// TIA Portal project "Trafik Işıkları Uygulaması 1" (V17)

(* hardware
DEVICE "S71500/ET200MP-Station_1"  S7-1500 station
   slot 0: "Profilschiene_0"  Rack  6ES7 590-1***0-0AA0
   slot 1: "PLC_1"  CPU 1518-4 PN/DP  6ES7 518-4AP00-0AB0  V2.9
      slot 3: "CPU-Display_1"  6ES7591-1BA00-0AA0
      slot 32768: "PROFINET-Schnittstelle_1"  X1
         slot 32769: "Port_1"  X1 P1
         slot 32770: "Port_2"  X1 P2
      slot 33024: "PROFINET interface_1"  X2
      slot 33280: "PROFINET interface GBIT_3"  X3
      slot 33536: "DP interface_1"  X4
      slot 34817: "Virtual CP interface port_1"  Virtual CP interface port  Virtual CP interface port
   slot 2: "AI 8xU/I/RTD/TC ST_1"  AI 8xU/I/RTD/TC ST  6ES7 531-7KF00-0AB0  V2.0
   slot 3: "AI 8xU/I/RTD/TC ST_2"  AI 8xU/I/RTD/TC ST  6ES7 531-7KF00-0AB0  V2.0
   slot 4: "AI 8xU/I/RTD/TC ST_3"  AI 8xU/I/RTD/TC ST  6ES7 531-7KF00-0AB0  V2.0
   slot 5: "AI 8xU/I/RTD/TC ST_4"  AI 8xU/I/RTD/TC ST  6ES7 531-7KF00-0AB0  V2.0
   slot 6: "DI 16x24VDC BA_1"  DI 16x24VDC BA  6ES7 521-1BH10-0AA0  V1.0
*)

// ===== PLC "PLC_1"  CPU 1518-4 PN/DP =====

VAR_GLOBAL   // PLC tag table "Standard-Variablentabelle"
   "START" AT %E0.0 : Bool;
   "A KIRMIZI" AT %A0.0 : Bool;
   "BAKIM" AT %E0.1 : Bool;
   "YARDIMCI KONTAK" AT %M0.0 : Bool;
   "Tag_2" AT %I0.2 : Bool;
   "DÖNGÜ" AT %M0.1 : Bool;
   "Tag_4" AT %T1 : Timer;
   "A SARI" AT %Q0.1 : Bool;
   "A YESİL" AT %Q0.2 : Bool;
   "B YESİL" AT %Q0.5 : Bool;
   "A YAYA Y" AT %Q0.7 : Bool;
   "B YAYA K" AT %Q1.0 : Bool;
   "B SARI" AT %Q0.4 : Bool;
   "B KIRMIZI" AT %Q0.3 : Bool;
   "B YAYA Y" AT %Q1.1 : Bool;
   "A YAYA K" AT %Q0.6 : Bool;
   "BAKIM YARDIMCI KONTAK" AT %M0.2 : Bool;
   "Clock_Byte" AT %MB50 : Byte;
   "Clock_10Hz" AT %M50.0 : Bool;
   "Clock_5Hz" AT %M50.1 : Bool;
   "Clock_2.5Hz" AT %M50.2 : Bool;
   "Clock_2Hz" AT %M50.3 : Bool;
   "Clock_1.25Hz" AT %M50.4 : Bool;
   "Clock_1Hz" AT %M50.5 : Bool;
   "Clock_0.625Hz" AT %M50.6 : Bool;
   "Clock_0.5Hz" AT %M50.7 : Bool;
   "Tag_1" AT %MD30 : Time;
   "Işık Süre" AT %QD30 : Time;
   "Tag_3" AT %QW30 : Word;
   "Tag_5" AT %MW30 : Word;
   "Tag_6" AT %ID30 : Time;
END_VAR

// folder: System blocks/Program resources

DATA_BLOCK "T1"   // DB1
{ S7_Optimized_Access := 'TRUE' }
AUTHOR : Simatic
FAMILY : IEC
NAME : IEC_TMR
VERSION : 1.0
// stored: InstanceOfName IEC_TIMER
"IEC_TIMER"
BEGIN
END_DATA_BLOCK

DATA_BLOCK "T2"   // DB2
{ S7_Optimized_Access := 'TRUE' }
AUTHOR : Simatic
FAMILY : IEC
NAME : IEC_TMR
VERSION : 1.0
// stored: InstanceOfName IEC_TIMER
"IEC_TIMER"
BEGIN
END_DATA_BLOCK

DATA_BLOCK "T3"   // DB3
{ S7_Optimized_Access := 'TRUE' }
AUTHOR : Simatic
FAMILY : IEC
NAME : IEC_TMR
VERSION : 1.0
// stored: InstanceOfName IEC_TIMER
"IEC_TIMER"
BEGIN
END_DATA_BLOCK

DATA_BLOCK "T4"   // DB5
{ S7_Optimized_Access := 'TRUE' }
AUTHOR : Simatic
FAMILY : IEC
NAME : IEC_TMR
VERSION : 1.0
// stored: InstanceOfName IEC_TIMER
"IEC_TIMER"
BEGIN
END_DATA_BLOCK

// folder: (top level)

FUNCTION "MHJ-PLC-Lab-Function-S71500" : Void   // FC9000, SCL
{ S7_Optimized_Access := 'TRUE' }
VERSION : 0.1
   VAR_TEMP
      Value : Byte;
      ForCounter : Int;
   END_VAR
   VAR CONSTANT
      Value_01_DW : DWord := 16#1223_5486;
      Value_02_DW : DWord := 16#A6C9_D1F5;
   END_VAR
BEGIN

   #Value:=PEEK(area := 16#82,
        dbNumber := 0,
        byteOffset := 511);
   #Value := #Value + 1;

   POKE(area := 16#82,
        dbNumber := 0,
        byteOffset := 511,
        value := #Value);

   POKE(area := 16#82,
        dbNumber := 0,
        byteOffset := 1016,
        value := #Value_01_DW);
   POKE(area := 16#82,
        dbNumber := 0,
        byteOffset := 1020,
        value := #Value_02_DW);

   FOR #ForCounter := 0 TO 63 DO
       #Value:=PEEK(area := 16#1,
            dbNumber := 0,
            byteOffset := #ForCounter);
       POKE(area := 16#81,
            dbNumber := 0,
            byteOffset := #ForCounter,
            value := #Value);
   END_FOR;
   #Value := PEEK(area := 16#1,
                  dbNumber := 0,
                  byteOffset := 512);
   POKE(area := 16#82,
        dbNumber := 0,
        byteOffset := 512,
        value := #Value);
END_FUNCTION

ORGANIZATION_BLOCK "Main"   // OB1, LAD, ProgramCycle
TITLE = "Main Program Sweep (Cycle)"
{ S7_Optimized_Access := 'TRUE' }
VERSION : 0.1
   VAR_INPUT
      Initial_Call : Bool;   // Initial call of this OB
      Remanence : Bool;   // =True, if remanent data are available
   END_VAR
   VAR_TEMP   // added for the SCL form of the ladder/FBD networks
      _w1 : Bool;
   END_VAR
BEGIN

REGION Network 1
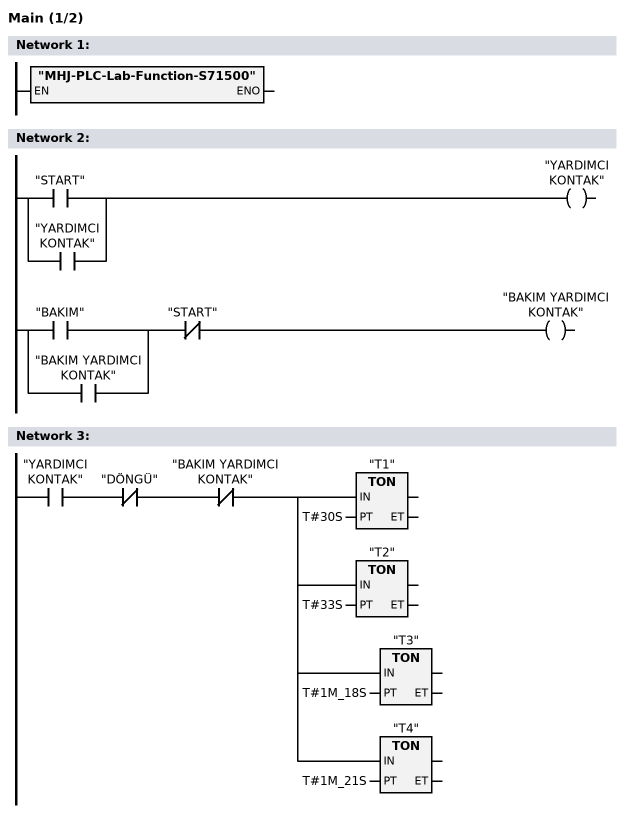
   RUNG wire#powerrail
      "MHJ-PLC-Lab-Function-S71500"()
   END_RUNG
   // the same network as SCL:
   "MHJ-PLC-Lab-Function-S71500"();
END_REGION

REGION Network 2
   RUNG wire#powerrail
      Contact( "START" )
      wire#w1
      Coil( "YARDIMCI KONTAK" )
   END_RUNG
   RUNG wire#powerrail
      Contact( "YARDIMCI KONTAK" )
   END_RUNG wire#w1
   RUNG wire#powerrail
      Contact( "BAKIM" )
      wire#w2
      I_Contact( "START" )
      Coil( "BAKIM YARDIMCI KONTAK" )
   END_RUNG
   RUNG wire#powerrail
      Contact( "BAKIM YARDIMCI KONTAK" )
   END_RUNG wire#w2
   // the same network as SCL:
   "YARDIMCI KONTAK" := "START" OR "YARDIMCI KONTAK";
   "BAKIM YARDIMCI KONTAK" := ("BAKIM" OR "BAKIM YARDIMCI KONTAK") AND NOT "START";
END_REGION

REGION Network 3
   #_w1 := "YARDIMCI KONTAK" AND NOT "DÖNGÜ" AND NOT "BAKIM YARDIMCI KONTAK";
   "T1".TON(IN := #_w1, PT := T#30S);
   "T2".TON(IN := #_w1, PT := T#33S);
   "T3".TON(IN := #_w1, PT := T#1M_18S);
   "T4".TON(IN := #_w1, PT := T#1M_21S);
END_REGION

REGION Network 4
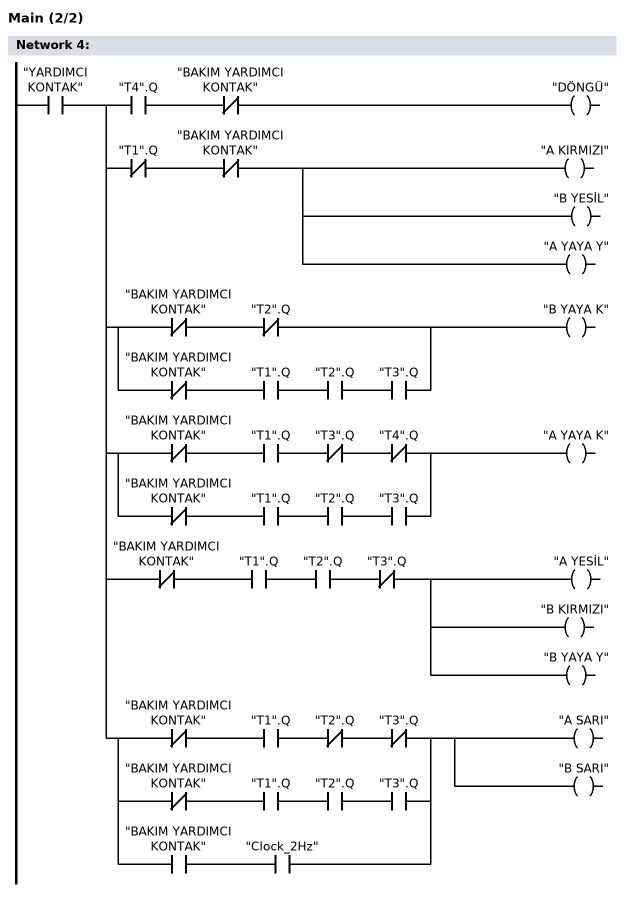
   RUNG wire#powerrail
      Contact( "YARDIMCI KONTAK" )
      wire#w1
      Contact( "T4".Q )
      I_Contact( "BAKIM YARDIMCI KONTAK" )
      Coil( "DÖNGÜ" )
   END_RUNG
   RUNG wire#w1
      I_Contact( "T1".Q )
      I_Contact( "BAKIM YARDIMCI KONTAK" )
      wire#w2
      Coil( "A KIRMIZI" )
   END_RUNG
   RUNG wire#w2
      Coil( "B YESİL" )
   END_RUNG
   RUNG wire#w2
      Coil( "A YAYA Y" )
   END_RUNG
   RUNG wire#w1
      I_Contact( "BAKIM YARDIMCI KONTAK" )
      I_Contact( "T2".Q )
      wire#w3
      Coil( "B YAYA K" )
   END_RUNG
   RUNG wire#w1
      I_Contact( "BAKIM YARDIMCI KONTAK" )
      Contact( "T1".Q )
      Contact( "T2".Q )
      Contact( "T3".Q )
   END_RUNG wire#w3
   RUNG wire#w1
      I_Contact( "BAKIM YARDIMCI KONTAK" )
      Contact( "T1".Q )
      I_Contact( "T3".Q )
      I_Contact( "T4".Q )
      wire#w4
      Coil( "A YAYA K" )
   END_RUNG
   RUNG wire#w1
      I_Contact( "BAKIM YARDIMCI KONTAK" )
      Contact( "T1".Q )
      Contact( "T2".Q )
      Contact( "T3".Q )
   END_RUNG wire#w4
   RUNG wire#w1
      I_Contact( "BAKIM YARDIMCI KONTAK" )
      Contact( "T1".Q )
      Contact( "T2".Q )
      I_Contact( "T3".Q )
      wire#w5
      Coil( "A YESİL" )
   END_RUNG
   RUNG wire#w5
      Coil( "B KIRMIZI" )
   END_RUNG
   RUNG wire#w5
      Coil( "B YAYA Y" )
   END_RUNG
   RUNG wire#w1
      I_Contact( "BAKIM YARDIMCI KONTAK" )
      Contact( "T1".Q )
      I_Contact( "T2".Q )
      I_Contact( "T3".Q )
      wire#w6
      Coil( "A SARI" )
   END_RUNG
   RUNG wire#w1
      I_Contact( "BAKIM YARDIMCI KONTAK" )
      Contact( "T1".Q )
      Contact( "T2".Q )
      Contact( "T3".Q )
   END_RUNG wire#w6
   RUNG wire#w1
      Contact( "BAKIM YARDIMCI KONTAK" )
      Contact( "Clock_2Hz" )
   END_RUNG wire#w6
   RUNG wire#w6
      Coil( "B SARI" )
   END_RUNG
   // the same network as SCL:
   "DÖNGÜ" := "YARDIMCI KONTAK" AND "T4".Q AND NOT "BAKIM YARDIMCI KONTAK";
   "A KIRMIZI" := "YARDIMCI KONTAK" AND NOT "T1".Q AND NOT "BAKIM YARDIMCI KONTAK";
   "B YESİL" := "A KIRMIZI";
   "A YAYA Y" := "A KIRMIZI";
   "B YAYA K" := "YARDIMCI KONTAK" AND ((NOT "BAKIM YARDIMCI KONTAK" AND NOT "T2".Q) OR (NOT "BAKIM YARDIMCI KONTAK" AND "T1".Q AND "T2".Q AND "T3".Q));
   "A YAYA K" := "YARDIMCI KONTAK" AND ((NOT "BAKIM YARDIMCI KONTAK" AND "T1".Q AND NOT "T3".Q AND NOT "T4".Q) OR (NOT "BAKIM YARDIMCI KONTAK" AND "T1".Q AND "T2".Q AND "T3".Q));
   "A YESİL" := "YARDIMCI KONTAK" AND NOT "BAKIM YARDIMCI KONTAK" AND "T1".Q AND "T2".Q AND NOT "T3".Q;
   "B KIRMIZI" := "A YESİL";
   "B YAYA Y" := "A YESİL";
   "A SARI" := "YARDIMCI KONTAK" AND ((NOT "BAKIM YARDIMCI KONTAK" AND "T1".Q AND NOT "T2".Q AND NOT "T3".Q) OR (NOT "BAKIM YARDIMCI KONTAK" AND "T1".Q AND "T2".Q AND "T3".Q) OR ("BAKIM YARDIMCI KONTAK" AND "Clock_2Hz"));
   "B SARI" := "A SARI";
END_REGION
END_ORGANIZATION_BLOCK